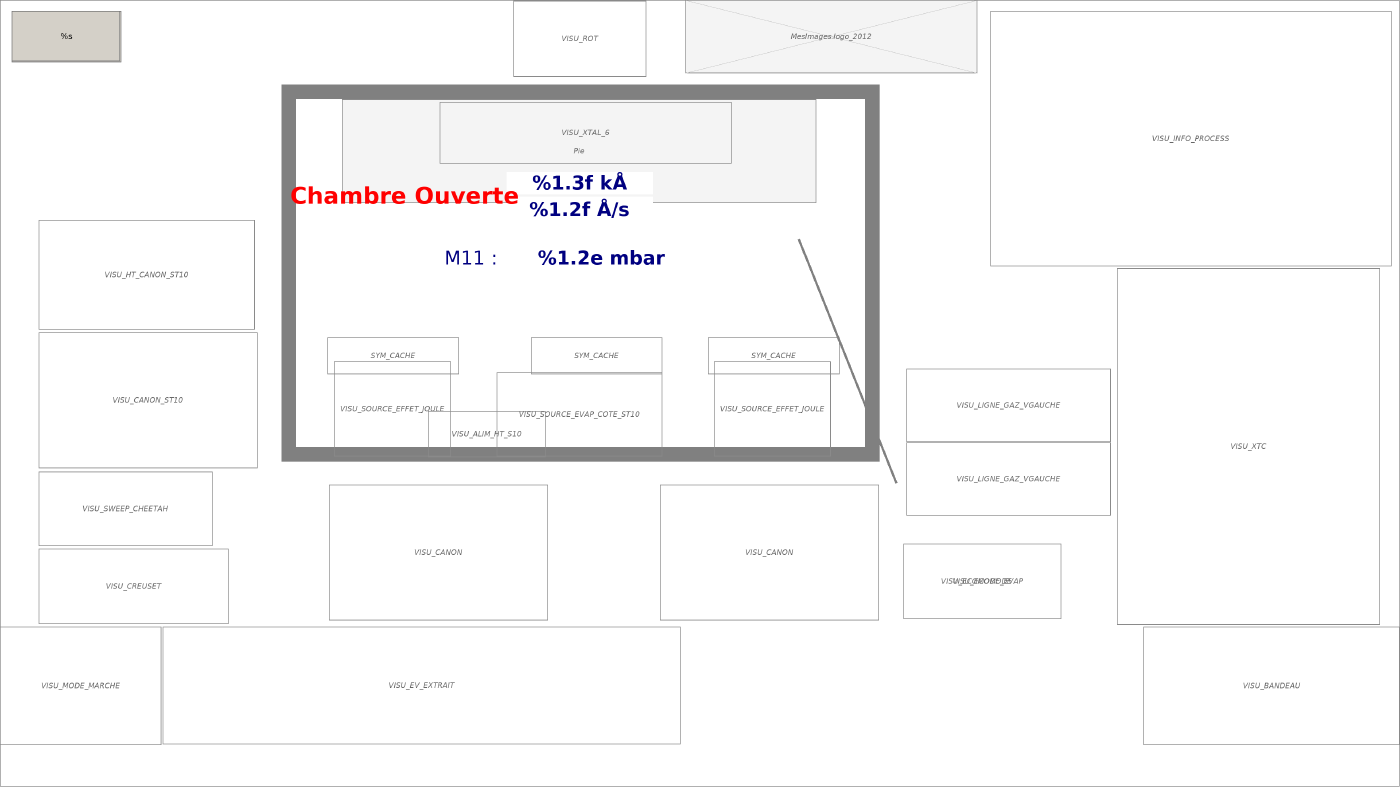
VISUALIZATION SYN_PROC  // 1920x1080, background image fond_blanc_1280_1024
    Frame (1239,746 216x103)
        shows VISU_ECOMODE()
    RoundedRectangle (386,116 820x517)
    Frame (704,1 182x104)
        shows VISU_ROT(m_Input_ROT := PRG_MOUVEMENT_PS.ROTATION_PS)
    Pie (469,136 650x142)
    Frame (223,860 710x161)
        shows VISU_EV_EXTRAIT()
    Frame (1568,860 352x162)
        shows VISU_BANDEAU(m_Input_MACHINE := Global_Variables.MACHINE)
    Rectangle (695,236 200x30), "%1.3f kÅ", text variable: PRG_EVAP.XTC3.STATE_Thickness
    Rectangle (695,270 200x35), "%1.2f Å/s", text variable: PRG_EVAP.XTC3.STATE_Rate
    Frame (0,860 221x162)
        shows VISU_MODE_MARCHE(m_Input_MACHINE := .MACHINE)
    Frame (603,140 400x84)
        shows VISU_XTAL_6(m_Input_XTAL := PRG_EVAP.QZ1, m_Input_NumFrame_Manu := 1)
    Button (16,15 150x70), "%s", text list: 'TextList_Navigation', text index: 0
        OnMouseClick: change screen: SYN_POMPAGE
    Frame (1532,368 360x489)
        shows VISU_XTC(M_Input_Evap := .PRG_EVAP.EVAPS1, M_Input_Ctrl := .PRG_EVAP.XTC3, M_Input_QZ1 := .PRG_EVAP.QZ1)
    Frame (1358,15 550x350), invisible if: NOT Global_Variables.MACHINE.STATE_Prod
        shows VISU_INFO_PROCESS()
    Frame (458,496 160x130)
        shows VISU_SOURCE_EFFET_JOULE(m_Input_SOURCE := PRG_EVAP.SOURCE2)
    Frame (451,665 300x186)
        shows VISU_CANON(m_Input_SOURCE := PRG_EVAP.SOURCE2)
    Frame (979,496 160x130)
        shows VISU_SOURCE_EFFET_JOULE(m_Input_SOURCE := PRG_EVAP.SOURCE3)
    Frame (905,665 300x186)
        shows VISU_CANON(m_Input_SOURCE := PRG_EVAP.SOURCE3)
    Frame (53,456 300x186)
        shows VISU_CANON_ST10(m_Input_SOURCE := .PRG_EVAP.SOURCE1)
    Frame (53,302 296x150)
        shows VISU_HT_CANON_ST10(m_Input_SOURCE := PRG_EVAP.SOURCE1)
    Frame (681,511 227x115)
        shows VISU_SOURCE_EVAP_COTE_ST10(m_Input_NO_IFIL_RET := FALSE, m_Input_NO_IEMISS_RET := FALSE, m_Input_SOURCE := PRG_EVAP.SOURCE1)
    Frame (728,463 180x50)
        shows SYM_CACHE(m_Input_CACHE := PRG_EVAP.CC11)
    Frame (971,463 180x50)
        shows SYM_CACHE(m_Input_CACHE := PRG_EVAP.CC13)
    Frame (449,463 180x50)
        shows SYM_CACHE(m_Input_CACHE := PRG_EVAP.CC12)
    Frame (587,564 161x63)
        shows VISU_ALIM_HT_S10(m_Input_HT := PRG_EVAP.SOURCE1)
    Rectangle (606,334 80x40), "M11 :"
    Rectangle (700,334 250x40), "%1.2e mbar", text variable: Global_Variables.PRG_POMPAGE.M11.STATE_Pression
    Polyline (1095,328)
    Polyline (1095,328) (1229,663)
    Polyline (1095,328)
    Polyline (1095,328)
    Frame (1243,607 280x100)
        shows VISU_LIGNE_GAZ_VGAUCHE(m_Input_MACHINE := MACHINE, m_Input_MASSFLOW := PRG_GAZ.DG[2], m_Input_LIGNE_GAZ := PRG_GAZ.LIGNE_GAZ[2])
    Frame (1243,506 280x100)
        shows VISU_LIGNE_GAZ_VGAUCHE(m_Input_MACHINE := MACHINE, m_Input_MASSFLOW := PRG_GAZ.DG[1], m_Input_LIGNE_GAZ := PRG_GAZ.LIGNE_GAZ[1])
    Frame (1239,746 216x103), invisible if: NOT MACHINE.STATE_Manu
        shows VISU_ECOMODE_EVAP()
    Label (390,237 330x63), "Chambre Ouverte", invisible if: PRG_POMPAGE.IN_FE11T
    Image (940,0 400x100), image: MesImages.logo_2012
    Frame (53,647 238x102)
        shows VISU_SWEEP_CHEETAH(m_Input_BALAYAGE := PRG_EVAP.SWEEP1)
    Frame (53,753 260x103)
        shows VISU_CREUSET(m_Input_CREUSET := PRG_EVAP.CRUCIBLE1, m_Input_NUM_CRUCIBLE := 1)
END_VISUALIZATION

(* stored: Version 1.1.0.1, ProductVersion 3.1.4026.18
   Visu SYN_PROC: Id {93d1845b-1462-4b07-a46d-f20d73f107f7} *)
